TYPE TankCtrl_Io_In :
STRUCT
	bNoWater		: BOOL;
	bOverload		: BOOL;
END_STRUCT
END_TYPE

(* stored: Version 1.1.0.1
   DUT TankCtrl_Io_In: Id {fa859c3e-9392-4634-b1e9-ddf067349c8a} *)
